FUNCTION EqualsLREAL : BOOL
VAR_INPUT
	n1 : LREAL;
	n2 : LREAL;
	epsilon : LREAL;
END_VAR

EqualsLREAL := ABS(n1 - n2) <= epsilon;

END_FUNCTION

(* stored: Version 1.1.0.1
   POU EqualsLREAL: Id {4aed6c8e-a7ce-0483-24c2-2e396af5ff43}, SpecialFunc None *)
